KUKA KRL program: SET_TOOL_FRAME.src

&ACCESS RVO1
&REL 1
&PARAM TEMPLATE = C:\KRC\Roboter\Template\FunctionVorgabe
&PARAM EDITMASK = *
DEFFCT BOOL SET_TOOL_FRAME( TOOL_NO:IN )

INT TOOL_NO

$STIFFNESS.TOOL = TOOL_DATA[TOOL_NO]
$STIFFNESS.COMMIT = TRUE

RETURN TRUE

ENDFCT
